(* IEC 61131-3 sources: plc_on_fpga_riscv_hybrid/RV_FPGA_PLC_IDE_Projects/PWM_DIM_ONE, 1 file *)

(* ---- PWM_DIM_ONE.il ---- *)
VAR
    Duty_Cycle   : UDINT
    PWM_1   : PWM
END_VAR

PROGRAM PWM_DIM_ONE
    DC :
        LD     %SW.0
        BOOL_TO_UDINT
        MUL    50
        ADD    50
        ST     Duty_Cycle
    PWM_Function_Block :
        CAL PWM_1(
            F  := 100,
            DC := Duty_Cycle,
            Q  => %LEDR.0)
END_PROGRAM
